// TwinCAT 3 PLC project tc_project_app
// ProgramVersion: 3.1.4023.0
// libraries:
//   Tc2_EtherCAT, * (Beckhoff Automation GmbH)
//   Tc2_MC2, * (Beckhoff Automation GmbH)
//   Tc2_Standard, * (Beckhoff Automation GmbH)
//   Tc2_SUPS, * (Beckhoff Automation GmbH)
//   Tc2_System, * (Beckhoff Automation GmbH)
//   Tc2_Utilities, * (Beckhoff Automation GmbH)
//   Tc3_MC2_AdvancedHoming, * (Beckhoff Automation GmbH)
//   Tc3_Module, * (Beckhoff Automation GmbH)
//   VisuDialogs, * (System)
// project tree:
//   / GlobalTextList.TcGTLO (not stored), NC_Task_1_SAF.TcTTO, PlcTask.TcTTO (not stored), Visualization Manager.TcVMO (not stored)
//   GVLs/ GVL_APP.TcGVL
//   POUs/Application_Specific/Applications/ Application_Template.TcPOU (not stored), SlitProg.TcPOU
//   POUs/Application_Specific/Axes/ Axis_Template.TcPOU (not stored), AXIS_1.TcPOU, AXIS_2.TcPOU, AXIS_3.TcPOU, AXIS_4.TcPOU, Pneumatics_Template.TcPOU (not stored)
//   POUs/ MAIN.TcPOU
//   tc_mca_std_lib/DUTs/Axis_Structures/ ST_AxisConfig.TcDUT (not stored), ST_AxisControl.TcDUT (not stored), ST_AxisDescription.TcDUT (not stored), ST_AxisError.TcDUT (not stored), ST_AxisInputs.TcDUT (not stored), ST_AxisPersistent.TcDUT (not stored), ST_AxisStatus.TcDUT (not stored), ST_AxisStruct.TcDUT (not stored), ST_GearAxis.TcDUT (not stored)
//   tc_mca_std_lib/DUTs/ E_AxisEngUnit.TcDUT (not stored), E_AxisLimitState.TcDUT (not stored), E_AxisParameters.TcTLEO (not stored), E_HomingRoutines.TcTLEO (not stored), E_AxisParameters.TcTLEO (not stored), E_MonitoringLedFunction.TcDUT (not stored), E_RestorePosition.TcDUT (not stored), E_SlitPairLimitState.TcDUT (not stored), I_Axis.TcIO (not stored), E_SlitPairStatesV2.TcDUT (not stored), E_SlitPairStates.TcDUT (not stored), ST_MonitoringAlarm.TcDUT (not stored), E_MotionFunctions.TcDUT (not stored), ST_McStatus.TcDUT (not stored)
//   tc_mca_std_lib/DUTs/Pneumatics/ E_PneumaticAxisErrors.TcDUT (not stored), E_PneumaticMode.TcDUT (not stored), ST_PneumaticAxisControl.TcDUT (not stored), ST_PneumaticAxisConfig.TcDUT (not stored), ST_PneumaticAxisInputs.TcDUT (not stored), ST_PneumaticAxisOutputs.TcDUT (not stored), ST_PneumaticAxisStatus.TcDUT (not stored), ST_PneumaticAxisStruct.TcDUT (not stored)
//   tc_mca_std_lib/GVLs/ GVL.TcGVL (not stored)
//   tc_mca_std_lib/POUs/ FB_ESSMonitoring.TcPOU (not stored)
//   tc_mca_std_lib/POUs/Motion/ FB_Axis.TcPOU (not stored), FB_Axis_1.TcPOU (not stored), FB_Axis_VirtualSlit.TcPOU (not stored), FB_SlitPair_ISIS.TcPOU (not stored)
//   tc_mca_std_lib/POUs/Motion/Homing/ FB_Homing.TcPOU (not stored), FB_Homing_1.TcPOU (not stored)
//   tc_mca_std_lib/POUs/Pneumatics/ FB_PneumaticAxis.TcPOU (not stored)
//   tc_mca_std_lib/VISUs/ languageSupport.TcTLO (not stored), MainVisu.TcVIS (not stored), ParameterTextList.TcTLO (not stored), PneumaticsVisu.TcVIS (not stored)
// real-time tasks:
//   TASK PlcTask: cycle T#10ms, priority 10, ADS port 351
// motion (NC):
//   TASK NC-Task 1 SAF: cycle T#2ms, priority 4, ADS port 501
//   TASK NC-Task 1 SVB: cycle T#10ms, priority 8, ADS port 511
//   AXIS Axis 1 (id 1)
//     OtherSettings: AllowMotionCmdToSlave=true
//     encoder EncType=1
//     drive DrvType=5
//       Analog: TorqueSetpointScale=10, ScaleFactorActTorque=0.1
//       TimeComp: TaskDelayCycles=1
//     controller CtrType=1
//       CtrPara: PriorControlFactor=1
//         Observer: BandWidth=20
//   AXIS Axis 2 (id 2)
//     OtherSettings: AllowMotionCmdToSlave=true
//     encoder EncType=1
//     drive DrvType=5
//       Analog: TorqueSetpointScale=10, ScaleFactorActTorque=0.1
//     controller CtrType=1
//       CtrPara: PriorControlFactor=1
//         Observer: BandWidth=20
//   AXIS Gap Size (id 3)
//     OtherSettings: AllowMotionCmdToSlave=true
//     encoder EncType=16
//       EncPara: MaxCount=#xffffffff
//     drive DrvType=5
//       Analog: VeloReferenz=1000, TorqueSetpointScale=10, ScaleFactorActTorque=0.1
//       TimeComp: TaskDelayCycles=1
//     controller CtrType=1
//       CtrPara: PriorControlFactor=1
//         Observer: BandWidth=20
//   AXIS Move Center (id 4)
//     OtherSettings: AllowMotionCmdToSlave=true
//     encoder EncType=16
//       EncPara: MaxCount=#xffffffff
//     drive DrvType=5
//       Analog: TorqueSetpointScale=10, ScaleFactorActTorque=0.1
//       TimeComp: TaskDelayCycles=1
//     controller CtrType=1
//       CtrPara: PriorControlFactor=1
//         Observer: BandWidth=20
// variable links:
//   tc_project_app Instance <-> NC-Task 1 SAF/Axes/Axis 1
//     PlcTask Inputs/GVL.astAxes[1].Axis.NcToPlc <-> Outputs/ToPlc
//     PlcTask Outputs/GVL.astAxes[1].Axis.PlcToNc <-> Inputs/FromPlc
//   tc_project_app Instance <-> NC-Task 1 SAF/Axes/Axis 2
//     PlcTask Inputs/GVL.astAxes[2].Axis.NcToPlc <-> Outputs/ToPlc
//     PlcTask Outputs/GVL.astAxes[2].Axis.PlcToNc <-> Inputs/FromPlc
//   tc_project_app Instance <-> NC-Task 1 SAF/Axes/Gap Size
//     PlcTask Inputs/GVL.astAxes[3].Axis.NcToPlc <-> Outputs/ToPlc
//     PlcTask Outputs/GVL.astAxes[3].Axis.PlcToNc <-> Inputs/FromPlc
//     PlcTask Outputs/SlitProg.mySlit.nGapSizeEncoder <-> Enc/Inputs/In/nDataIn1
//   tc_project_app Instance <-> NC-Task 1 SAF/Axes/Move Center
//     PlcTask Inputs/GVL.astAxes[4].Axis.NcToPlc <-> Outputs/ToPlc
//     PlcTask Outputs/GVL.astAxes[4].Axis.PlcToNc <-> Inputs/FromPlc
//     PlcTask Outputs/SlitProg.mySlit.nGapCentreEncoder <-> Enc/Inputs/In/nDataIn1

CONFIGURATION tc_project_app
    RESOURCE PLC ON TwinCAT3
        TASK NC_Task_1_SAF(INTERVAL := T#2ms, PRIORITY := 4);
    END_RESOURCE
END_CONFIGURATION

// ---- GVLs/GVL_APP.TcGVL
{attribute 'qualified_only'}
VAR_GLOBAL
END_VAR

VAR_GLOBAL CONSTANT
    nAXIS_NUM: UINT := 4;
    nPNEUMATIC_AXIS_NUM: UINT := 0;
END_VAR

// ---- POUs/Application_Specific/Applications/SlitProg.TcPOU
PROGRAM SlitProg
VAR_INPUT
    mySlit : FB_SlitPair_ISIS;
   
END_VAR

(*SETUP INSTRUCTIONS
    All Axes:
        Allow motion commands to external setpoint axis := FALSE;

    Virtual axes:
        Dynamics of virtual axes must be configured considering coupled mechanicals (e.g. don't set velocities your real axes can't achieve)
*)
mySlit.nIdPositiveAxis := 1;
mySlit.nIdNegativeAxis := 2;
mySlit.nIdGapSizeAxis := 3;
mySlit.nIdGapCentreAxis :=4;
mySlit();

END_PROGRAM

// ---- POUs/Application_Specific/Axes/AXIS_1.TcPOU
PROGRAM AXIS_1
VAR
//Outputs: Power for Limit switches, Home Sensors, etc.
    //bPowerSwitchesAxis1 AT %Q*: BOOL:= TRUE;

//Hardware interlocks
    //bInterlockFwdOK AT %I*: BOOL;
END_VAR

//Initial parameters of an Axis
(*IF _TaskInfo[fbGetCurTaskIndex.index].FirstCycle THEN
    //Axis description for EPICS PV
    GVL.astAxes[1].stDescription.sAxisName := 'MotorApplication1';
    GVL.astAxes[1].stDescription.eUnit := E_AxisEngUnit.eMeter;
    GVL.astAxes[1].stDescription.nPrefix := -3;

    //Initial default values:
    GVL.astAxes[1].stConfig.eHomeSeq := 0;
    GVL.astAxes[1].stConfig.fHomePosition := 0.0;
    GVL.astAxes[1].stConfig.fHomeFinishDistance := 0.0;
    GVL.astAxes[1].stConfig.eRestorePosition := E_RestorePosition.eRestoreWithoutHome;
END_IF*)

//Define ACTIONS() or write exclusive code for an specific axis.
(*Eg. Stop when temperature reaches certain values, reduce speed if  a signal is activated, etc.
Eg. GVL.astAxes[x].stControl.bInterlockFwd := NOT bInterlockFwdOK;*)

//Limits for positive axis, Axis 1
IF astAxes[1].stStatus.fActPosition > 100 THEN
    SlitProg.mySlit.bPositiveAxis_FwdLimit := FALSE;
ELSE
     SlitProg.mySlit.bPositiveAxis_FwdLimit :=TRUE;
END_IF
IF astAxes[1].stStatus.fActPosition < -100 THEN
     SlitProg.mySlit.bPositiveAxis_BwdLimit :=FALSE;
ELSE
     SlitProg.mySlit.bPositiveAxis_BwdLimit :=TRUE;
END_IF

END_PROGRAM

// ---- POUs/Application_Specific/Axes/AXIS_2.TcPOU
PROGRAM AXIS_2
VAR
//Outputs: Power for Limit switches, Home Sensors, etc.
    //bPowerSwitchesAxis1 AT %Q*: BOOL:= TRUE;

//Hardware interlocks
    //bInterlockFwdOK AT %I*: BOOL;
END_VAR

//Initial parameters of an Axis
(*IF _TaskInfo[fbGetCurTaskIndex.index].FirstCycle THEN
    //Axis description for EPICS PV
    GVL.astAxes[1].stDescription.sAxisName := 'MotorApplication1';
    GVL.astAxes[1].stDescription.eUnit := E_AxisEngUnit.eMeter;
    GVL.astAxes[1].stDescription.nPrefix := -3;

    //Initial default values:
    GVL.astAxes[1].stConfig.eHomeSeq := 0;
    GVL.astAxes[1].stConfig.fHomePosition := 0.0;
    GVL.astAxes[1].stConfig.fHomeFinishDistance := 0.0;
    GVL.astAxes[1].stConfig.eRestorePosition := E_RestorePosition.eRestoreWithoutHome;
END_IF*)

//Define ACTIONS() or write exclusive code for an specific axis.
(*Eg. Stop when temperature reaches certain values, reduce speed if  a signal is activated, etc.
Eg. GVL.astAxes[x].stControl.bInterlockFwd := NOT bInterlockFwdOK;*)

//Limits for negative axis, Axis 2
IF astAxes[2].stStatus.fActPosition > 100 THEN
    SlitProg.mySlit.bNegativeAxis_FwdLimit := FALSE;
ELSE
     SlitProg.mySlit.bNegativeAxis_FwdLimit :=TRUE;
END_IF
IF astAxes[2].stStatus.fActPosition < -100 THEN
     SlitProg.mySlit.bNegativeAxis_BwdLimit :=FALSE;
ELSE
     SlitProg.mySlit.bNegativeAxis_BwdLimit :=TRUE;
END_IF

END_PROGRAM

// ---- POUs/Application_Specific/Axes/AXIS_3.TcPOU
PROGRAM AXIS_3
VAR
//Outputs: Power for Limit switches, Home Sensors, etc.
    //bPowerSwitchesAxis1 AT %Q*: BOOL:= TRUE;

//Hardware interlocks
    //bInterlockFwdOK AT %I*: BOOL;
END_VAR

//Initial parameters of an Axis
(*IF _TaskInfo[fbGetCurTaskIndex.index].FirstCycle THEN
    //Axis description for EPICS PV
    GVL.astAxes[1].stDescription.sAxisName := 'MotorApplication1';
    GVL.astAxes[1].stDescription.eUnit := E_AxisEngUnit.eMeter;
    GVL.astAxes[1].stDescription.nPrefix := -3;

    //Initial default values:
    GVL.astAxes[1].stConfig.eHomeSeq := 0;
    GVL.astAxes[1].stConfig.fHomePosition := 0.0;
    GVL.astAxes[1].stConfig.fHomeFinishDistance := 0.0;
    GVL.astAxes[1].stConfig.eRestorePosition := E_RestorePosition.eRestoreWithoutHome;
END_IF*)

//Define ACTIONS() or write exclusive code for an specific axis.
(*Eg. Stop when temperature reaches certain values, reduce speed if  a signal is activated, etc.
Eg. GVL.astAxes[x].stControl.bInterlockFwd := NOT bInterlockFwdOK;*)

END_PROGRAM

// ---- POUs/Application_Specific/Axes/AXIS_4.TcPOU
PROGRAM AXIS_4
VAR
//Outputs: Power for Limit switches, Home Sensors, etc.
    //bPowerSwitchesAxis1 AT %Q*: BOOL:= TRUE;

//Hardware interlocks
    //bInterlockFwdOK AT %I*: BOOL;
END_VAR

//Initial parameters of an Axis
(*IF _TaskInfo[fbGetCurTaskIndex.index].FirstCycle THEN
    //Axis description for EPICS PV
    GVL.astAxes[1].stDescription.sAxisName := 'MotorApplication1';
    GVL.astAxes[1].stDescription.eUnit := E_AxisEngUnit.eMeter;
    GVL.astAxes[1].stDescription.nPrefix := -3;

    //Initial default values:
    GVL.astAxes[1].stConfig.eHomeSeq := 0;
    GVL.astAxes[1].stConfig.fHomePosition := 0.0;
    GVL.astAxes[1].stConfig.fHomeFinishDistance := 0.0;
    GVL.astAxes[1].stConfig.eRestorePosition := E_RestorePosition.eRestoreWithoutHome;
END_IF*)

//Define ACTIONS() or write exclusive code for an specific axis.
(*Eg. Stop when temperature reaches certain values, reduce speed if  a signal is activated, etc.
Eg. GVL.astAxes[x].stControl.bInterlockFwd := NOT bInterlockFwdOK;*)

END_PROGRAM

// ---- POUs/MAIN.TcPOU
PROGRAM MAIN
VAR
    sVersion: STRING := '1.0.0';
    aIAxes: ARRAY [1..GVL_APP.nAXIS_NUM] OF I_Axis;
    afbAxes: ARRAY [1..GVL_APP.nAXIS_NUM] OF FB_Axis;
    afbPneumaticAxes: ARRAY [1..GVL_APP.nPNEUMATIC_AXIS_NUM] OF FB_PneumaticAxis;
    hmiAxisSelection: INT := 1; //Not possible to use local hmi variables for array indexes
    hmiPneumaticAxisSelection: INT := 1;
//Startup, Shutdown and UPS
    fbUPS: FB_S_UPS_CX51x0;
    eUpsMode: E_S_UPS_Mode := eSUPS_WrPersistData_Shutdown;
    eStartUp: (eColdStart, eReadAxisFeedbackType, eCheckReadDone, eExecuteRestore, eCheckRestore, eFinishRestore);
    bPositionRestoreDone: BOOL := FALSE;
    bRestoreExecute: BOOL := FALSE;
    bExecuteReadEncRefSys: BOOL := FALSE;
    nRetry: INT;
    iAxes: UINT; //index for for loops in Position recovery actions
    afbReadEncRefSys: ARRAY [1..GVL_APP.nAXIS_NUM] OF MC_ReadParameter;
    afbSetPosition: ARRAY [1..GVL_APP.nAXIS_NUM] OF MC_SetPosition;
    afbReadPositionBias: ARRAY [1..GVL_APP.nAXIS_NUM] OF MC_ReadParameter;
    afbWritePositionBias: ARRAY [1..GVL_APP.nAXIS_NUM] OF MC_WriteParameter;
    fbGetDeviceIdentification: FB_GetDeviceIdentificationEx;
END_VAR

VAR PERSISTENT
    bRestoreOnStartup: BOOL;
END_VAR

POSITION_RECOVERY();
PROG();
AXES();

ACTION AXES:
//First cycle, assign FB_axis to interface array
IF _TaskInfo[fbGetCurTaskIndex.index].FirstCycle THEN
    FOR GVL.iAxis := 1 TO GVL_APP.nAXIS_NUM DO
        afbAxes[GVL.iAxis].stAxis REF= astAxes[GVL.iAxis];
        aIAxes[GVL.iAxis] := afbAxes[GVL.iAxis];
    END_FOR
    //Custom axis types defined and linked to aiAxes here
      //FB_CustomAxis extends FB_axis
        //fbCustomAxis.stAxis REF= astAxes[x];
        //aIAxes[x] := fbCustomAxis;
END_IF

//Execute FB_Axis logic
FOR GVL.iAxis := 1 TO GVL_APP.nAXIS_NUM DO
    aIAxes[GVL.iAxis].Run();
END_FOR

//Execute Pneumatic Axis logic
FOR GVL.iPneumaticAxis := 1 TO GVL_APP.nPNEUMATIC_AXIS_NUM DO
    afbPneumaticAxes[GVL.iPneumaticAxis](stPneumaticAxisStruct := GVL.astPneumaticAxes[GVL.iPneumaticAxis]);
END_FOR
END_ACTION

ACTION CHECK_UPS:
fbUPS(eUpsMode := eUpsMode);

FOR iAxes := 1 TO GVL_APP.nAXIS_NUM DO
    //Read encoder position BIAS
    IF astAxes[iAxes].stStatus.bAxisInitialized THEN
        afbReadPositionBias[iAxes](Axis := GVL.astAxes[iAxes].Axis,
                        Enable := TRUE,
                        ReadMode:= READMODE_CYCLIC,
                        ParameterNumber := E_AxisParameters.AxisEncoderOffset);
    END_IF
END_FOR

IF eGlobalSUpsState = eSUPS_PowerFailure THEN
    //first cycle of powerfailure
    //execute code that should only be done once with each powerfailure, i.e. increase powerfailure counter
    bRestoreOnStartup := TRUE;
    STORE_PERSISTENT();
    RETURN;
ELSIF eGlobalSUpsState <> eSUPS_PowerOK THEN
    //next cycles of powerfailure
    //skip regular code execution for the remaining cycles of the powerfailure/writing of persistent data/quick shutdown...
    RETURN;
END_IF
END_ACTION

ACTION POSITION_RECOVERY:
fbGetDeviceIdentification(bExecute := TRUE);
IF (fbGetDeviceIdentification.stDevIdent.strHardwareSerialNo <> '') THEN
    CHECK_UPS();
    RESTORE_POSITIONS();
END_IF
END_ACTION

ACTION PROG:
//Get task index for Axes parameters initialization.
GVL.fbGetCurTaskIndex();

//Call the programs that are defined in the "Application Specific" folder.
//Create as many programs in that folder as axes and applications you have or need

//Axes initial parameters and program
//Axis_Template();
//Pneumatics_Template();

//Application program calls
//Application_Template();

AXIS_1();
AXIS_2();
AXIS_3();
AXIS_4();

SlitProg();
END_ACTION

ACTION RESTORE_POSITIONS:
//This ACT will restore the position of an incremental axis on startup with the act position it read before losing power.
//It checks the type of axis, 0=incremental, and that the axis was stationary at shut down.
//Because 0 equates to incremental we also need to check that the data is valid, otherwise by default it would restore all axes.
//By default an axis will not restore the position unless it is set to opt-in, i.e. GVL.aAxes[iAxes].stConfig.eRestorePosition is non-zero.
//This needs to be initialised somewhere in TwinCAT code otherwise it will not be available at start up.
//A restore will only be performed on a loss of power, this code shouldn't make any changes on a reset cold, a rest origin or a download.
//There is a enum to allow for different types of restore modes, currently only one is implemented.
//0 'DontRestore'
//1 'RestoreWithoutHome' -restores the position using a set position fb and does not set the home bit in the axis struct.
//Note from Beckhoff: "A maximum of 1 MB persistent data can be reliably saved over the entire service life."
//Encoder Reference system types: https://infosys.beckhoff.com/english.php?content=../content/1033/tf50x0_tc3_nc_ptp/3439907723.html&id=
//INCREMENTAL=0;
//ABSOLUTE=1;
//ABSOLUTE (modulo)=2;
//ABSOLUTE MULTITURN RANGE (with single overflow)=3;
//INCREMENTAL (singleturn absolute)=4;
//ABSOLUTE SINGLETURN RANGE (with single overflow)=5;


IF bRestoreOnStartup AND eGlobalSUpsState = eSUPS_PowerOK THEN
    bRestoreOnStartup := FALSE;
    bRestoreExecute := TRUE;
END_IF

//Upon startup bPositionRestoreDone will be set to FALSE, after successfully completing the following code it will be set TRUE
//and should stay TRUE for the rest of the time the PLC is operational, thus this routine should only be completed once.
IF bRestoreExecute AND NOT bPositionRestoreDone THEN
    //Cycle through function blocks that read the encoder reference system i.e. whether axis is incremental or absolute
    FOR iAxes := 1 TO GVL_APP.nAXIS_NUM DO
         afbReadEncRefSys[iAxes](
            Axis := GVL.astAxes[iAxes].Axis,
            ParameterNumber := MC_AxisParameter.AxisEncoderReferenceSystem,
            ReadMode := E_READMODE.READMODE_ONCE);
    END_FOR

    //Cycle through set position and MC_WritePArameter function blocks for each axis
    FOR iAxes := 1 TO GVL_APP.nAXIS_NUM DO
        afbSetPosition[iAxes](
            Axis := GVL.astAxes[iAxes].Axis,
            Position := astAxesPersistent[iAxes].fPositionAtShutdown);

        afbWritePositionBias[iAxes](
            Axis:= GVL.astAxes[iAxes].Axis,
            ParameterNumber:= E_AxisParameters.AxisEncoderOffset,
            Value:= astAxesPersistent[iAxes].fEncoderBiasAtShutdown);
    END_FOR

    CASE eStartUp OF
        eColdStart:
            //First cycle of the PLC, do nothing just give one cycle for variables to initialise
            IF NOT bPositionRestoreDone THEN
                eStartUp := eReadAxisFeedbackType;
                nRetry := 0;
            END_IF

        eReadAxisFeedbackType:
            //Exectute the function blocks to read the encoder reference system (0=inc OR 1=ABS)
            FOR iAxes := 1 TO GVL_APP.nAXIS_NUM DO
                afbReadEncRefSys[iAxes].Enable := TRUE;
                eStartUp := eCheckReadDone;
            END_FOR

        eCheckReadDone:
            //Check the encoder reference system has been read for all axis -> if busy then continue with PLC cycle and check again next time.
            //If afbReadEncRefSys not started then go back a step.
            //If any axes result in an error the code will get stuck here, this happens if GVL_APP.nAXIS_NUM is not set correctly
            FOR iAxes := 1 TO GVL_APP.nAXIS_NUM DO
                IF NOT afbReadEncRefSys[iAxes].Valid THEN
                    IF afbReadEncRefSys[iAxes].Busy THEN
                        //Exit MAIN.STARTUP Action and wait till next cycle, needs to cycle through whole program in order for data to update
                        RETURN;
                    ELSE
                        //Sometimes the code gets here and the afbReadEncRefSys[iAxes] misses the rising edge. If  the code gets here it means
                        //valid=FALSE and .busy=FALSE which indicateds the FB probably hasn't started and thus needs to see a rising edge.
                        //Set execute to low, Exit MAIN.STARTUP and go back a step in the CASE statement.
                        afbReadEncRefSys[iAxes].Enable := FALSE;
                        eStartUp := eReadAxisFeedbackType;
                        nRetry := nRetry + 1; //counter used for troubleshooting to see how many cycles it takes before afbReadEncRefSys function blocks are read correctly
                        RETURN;
                    END_IF
                END_IF
            END_FOR
            //If the code gets here all axes have .valid=TRUE for all axes
            eStartUp := eExecuteRestore;

        eExecuteRestore:
            //Execute position and encoder BIAS restore by setting Execute = TRUE
           FOR iAxes := 1 TO GVL_APP.nAXIS_NUM DO
                IF GVL.astAxes[iAxes].stConfig.eRestorePosition = E_RestorePosition.eRestoreWithoutHome THEN
                    //Restore position value for incremental encoders
                    IF NOT astAxesPersistent[iAxes].bMovingAtShutdown AND
                    (afbReadEncRefSys[iAxes].Value = 0 OR
                     afbReadEncRefSys[iAxes].Value = 2 OR
                     afbReadEncRefSys[iAxes].Value = 4) THEN
                       afbSetPosition[iAxes].Execute := TRUE;
                    //Restore encoder position BIAS for absolute encoders
                    ELSIF afbReadEncRefSys[iAxes].Value = 1 OR
                    afbReadEncRefSys[iAxes].Value = 3 OR
                    afbReadEncRefSys[iAxes].Value = 5 THEN
                       afbWritePositionBias[iAxes].Execute := TRUE;
                    END_IF
                ELSE
                    RETURN;
                END_IF
            END_FOR
            eStartUp := eCheckRestore;


        eCheckRestore:
            //Check the set position and write enocder BIAS fbs are finished
            //Nothing actually happens if the restore is not done, the code just returns from here each cycle and the
            //bPositionRestoreDone will never get set to TRUE and will take up cycle time
            FOR iAxes := 1 TO GVL_APP.nAXIS_NUM DO
                IF GVL.astAxes[iAxes].stConfig.eRestorePosition = E_RestorePosition.eRestoreWithoutHome THEN
                    IF NOT astAxesPersistent[iAxes].bMovingAtShutdown AND
                    (afbReadEncRefSys[iAxes].Value = 0 OR
                     afbReadEncRefSys[iAxes].Value = 2 OR
                     afbReadEncRefSys[iAxes].Value = 4) THEN
                        IF NOT afbSetPosition[iAxes].Done THEN
                            afbSetPosition[iAxes].Execute := FALSE;
                            eStartUp := eExecuteRestore;
                            RETURN;
                        END_IF
                     ELSIF afbReadEncRefSys[iAxes].Value = 1 OR
                     afbReadEncRefSys[iAxes].Value = 3 OR
                     afbReadEncRefSys[iAxes].Value = 5 THEN
                        IF NOT afbWritePositionBias[iAxes].Done THEN
                            afbWritePositionBias[iAxes].Execute := FALSE;
                            eStartUp := eExecuteRestore;
                            RETURN;
                        END_IF
                    END_IF
                ELSE
                    RETURN;
                END_IF
            END_FOR
            eStartUp :=  eFinishRestore;

        eFinishRestore:
            //Remove execute = TRUE for afbRestorePosition and fbWritePositionBias
            FOR iAxes := 1 TO GVL_APP.nAXIS_NUM DO
                afbSetPosition[iAxes].Execute := FALSE;
                afbWritePositionBias[iAxes].Execute := FALSE;
                bPositionRestoreDone := TRUE;
                bRestoreExecute := FALSE;
            END_FOR
    END_CASE
END_IF
END_ACTION

ACTION STORE_PERSISTENT:
FOR iAxes := 1 TO GVL_APP.nAXIS_NUM DO
    //Store Position beofre shutdown
    astAxesPersistent[iAxes].fPositionAtShutdown := GVL.astAxes[iAxes].Axis.NcToPlc.ActPos;

    //Store encoder position BIAS at shutdown
    astAxesPersistent[iAxes].fEncoderBiasAtShutdown := afbReadPositionBias[iAxes].Value;

    //Store value of moving at shutdown
    IF GVL.astAxes[iAxes].Axis.Status.StandStill OR GVL.astAxes[iAxes].Axis.Status.Disabled THEN
        astAxesPersistent[iAxes].bMovingAtShutdown := FALSE;
    ELSE
        astAxesPersistent[iAxes].bMovingAtShutdown := TRUE;
    END_IF
END_FOR
END_ACTION

END_PROGRAM
